# EPICS autosave request: cmds/auto_settings.req
file "spinnaker_settings.req",            P=$(P),  R=$(R)
file "NDStdArrays_settings.req",          P=$(P),  R=$(R)
file "commonPlugin_settings.req",         P=$(P)
